// TIA Portal project "Manufacturing Line Assembly" (V17)
// Manufacturing Line Assembly
// Product should move through 3 assembly stations, with each station operating for 15s.

(* hardware
DEVICE "S7-1200 station_1"  S7-1200 Station
   slot 0: "Rack_0"  S7-1200 Rack  Rack  V1.0
   slot 1: "PLC_1"  CPU 1215FC DC/DC/RLY  6ES7 215-1HF40-0XB0  V4.5
*)

// ===== PLC "PLC_1"  CPU 1215FC DC/DC/RLY =====

VAR_GLOBAL   // PLC tag table "Default tag table"
   "Sensor_1" AT %I0.0 : Bool;
   "Sensor_2" AT %I0.1 : Bool;
   "Sensor_3" AT %I0.2 : Bool;
   "Start_Button" AT %I0.3 : Bool;
   "Station_1" AT %Q0.0 : Bool;
   "Station_2" AT %Q0.1 : Bool;
   "Station_3" AT %Q0.2 : Bool;
   "Conveyor" AT %Q0.3 : Bool;
END_VAR

// folder: System blocks/Program resources

DATA_BLOCK "IEC_Timer_0_DB"   // DB2
{ S7_Optimized_Access := 'TRUE' }
AUTHOR : Simatic
FAMILY : IEC
NAME : IEC_TMR
VERSION : 1.0
// stored: InstanceOfName IEC_TIMER
"IEC_TIMER"
BEGIN
END_DATA_BLOCK

DATA_BLOCK "IEC_Timer_0_DB_1"   // DB3
{ S7_Optimized_Access := 'TRUE' }
AUTHOR : Simatic
FAMILY : IEC
NAME : IEC_TMR
VERSION : 1.0
// stored: InstanceOfName IEC_TIMER
"IEC_TIMER"
BEGIN
END_DATA_BLOCK

DATA_BLOCK "IEC_Timer_0_DB_2"   // DB4
{ S7_Optimized_Access := 'TRUE' }
AUTHOR : Simatic
FAMILY : IEC
NAME : IEC_TMR
VERSION : 1.0
// stored: InstanceOfName IEC_TIMER
"IEC_TIMER"
BEGIN
END_DATA_BLOCK

// folder: (top level)

ORGANIZATION_BLOCK "Main"   // OB1, LAD, ProgramCycle
TITLE = "Main Program Sweep (Cycle)"
{ S7_Optimized_Access := 'TRUE' }
VERSION : 0.1
   VAR_INPUT
      Initial_Call : Bool;   // Initial call of this OB
      Remanence : Bool;   // =True, if remanent data are available
   END_VAR
BEGIN

REGION Network 1
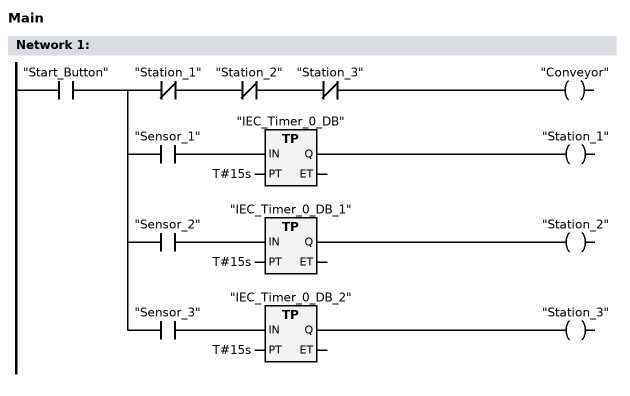
   "Conveyor" := "Start_Button" AND NOT "Station_1" AND NOT "Station_2" AND NOT "Station_3";
   "IEC_Timer_0_DB".TP(IN := "Start_Button" AND "Sensor_1", PT := T#15s);
   "Station_1" := "IEC_Timer_0_DB".Q;
   "IEC_Timer_0_DB_1".TP(IN := "Start_Button" AND "Sensor_2", PT := T#15s);
   "Station_2" := "IEC_Timer_0_DB_1".Q;
   "IEC_Timer_0_DB_2".TP(IN := "Start_Button" AND "Sensor_3", PT := T#15s);
   "Station_3" := "IEC_Timer_0_DB_2".Q;
END_REGION
END_ORGANIZATION_BLOCK